// TwinCAT 3 PLC project Crane
// ProgramVersion: 3.1.4026.11
// libraries:
//   Tc2_Standard, * (Beckhoff Automation GmbH)
//   Tc2_System, * (Beckhoff Automation GmbH)
//   [Resi4MPM], * (Jan Wilch)
//   [xPPU], * (Jan Wilch)
// project tree:
//   / HardwareContainer.TcPOU, MAIN.TcPOU, PlcTask.TcTTO
// real-time tasks:
//   TASK PlcTask: cycle T#10ms, priority 20, ADS port 350
//   TASK PlcTask1: cycle T#10ms, priority 23, ADS port 351
//   TASK PlcTask2: cycle T#10ms, priority 22, ADS port 352
//   TASK PlcTask3: cycle T#10ms, priority 21, ADS port 353
// I/O:
//   DEVICE Device (EtherCAT), AmsNetId 192.168.82.13.3.1
//     Term 84 (EK1200) [EK1200-5000 EtherCAT Netzteil (2A E-Bus)]
//       Klemme 2 (EK1110) [EK1110 EtherCAT-Verlängerung]
//     BK1 (EK1100) [EK1100 EtherCAT-Koppler (2A E-Bus)]
//       1.2 (EL1004) [EL1004 4K. Dig. Eingang 24V, 3ms]
//       1.3 (EL1004) [EL1004 4K. Dig. Eingang 24V, 3ms]
//       1.4 (EL1004) [EL1004 4K. Dig. Eingang 24V, 3ms]
//       1.5 (EL1004) [EL1004 4K. Dig. Eingang 24V, 3ms]
//       1.6 (EL2004) [EL2004 4K. Dig. Ausgang 24V, 0.5A]
//       1.9 (EL2004) [EL2004 4K. Dig. Ausgang 24V, 0.5A]
//       1.10 (EL2004) [EL2004 4K. Dig. Ausgang 24V, 0.5A]
//       1.11 (EL2004) [EL2004 4K. Dig. Ausgang 24V, 0.5A]
//       1.12 (EL1004) [EL1004 4K. Dig. Eingang 24V, 3ms]
//       1.13 (EL3162) [EL3162 2K. Ana. Eingang 0-10V]
//       1.14 (EL9011) [EL9011 Endklemme]
//     BK2&3 (EK1100) [EK1100 EtherCAT-Koppler (2A E-Bus)]
//       2&3.2 (EL1004) [EL1004 4K. Dig. Eingang 24V, 3ms]
//       2&3.3 (EL1004) [EL1004 4K. Dig. Eingang 24V, 3ms]
//       2&3.4 (EL1004) [EL1004 4K. Dig. Eingang 24V, 3ms]
//       2&3.5 (EL1004) [EL1004 4K. Dig. Eingang 24V, 3ms]
//       2&3.6 (EL1004) [EL1004 4K. Dig. Eingang 24V, 3ms]
//       2&3.7 (EL1004) [EL1004 4K. Dig. Eingang 24V, 3ms]
//       2&3.10 (EL2004) [EL2004 4K. Dig. Ausgang 24V, 0.5A]
//       2&3.11 (EL2004) [EL2004 4K. Dig. Ausgang 24V, 0.5A]
//       2&3.12 (EL2004) [EL2004 4K. Dig. Ausgang 24V, 0.5A]
//       2&3.13 (EL2004) [EL2004 4K. Dig. Ausgang 24V, 0.5A]
//       2&3.14 (EL1004) [EL1004 4K. Dig. Eingang 24V, 3ms]
//       2&3.16 (EL4102) [EL4102 2K. Ana. Ausgang 0-10V]
//       2&3.17 (EL4102) [EL4102 2K. Ana. Ausgang 0-10V]
//       2&3.18 (EL9011) [EL9011 Endklemme]
//     BK4 (EK1100) [EK1100 EtherCAT-Koppler (2A E-Bus)]
//       4.2 (EL1808) [EL1808 8K. Dig. Eingang 24V, 3ms]
//       4.3 (EL1004) [EL1004 4K. Dig. Eingang 24V, 3ms]
//       4.4 (EL1004) [EL1004 4K. Dig. Eingang 24V, 3ms]
//       4.5 (EL1004) [EL1004 4K. Dig. Eingang 24V, 3ms]
//       4.6 (EL1004) [EL1004 4K. Dig. Eingang 24V, 3ms]
//       4.7 (EL1004) [EL1004 4K. Dig. Eingang 24V, 3ms]
//       4.8 (EL3064) [EL3064 4K.Ana. Eingang 0-10V]
//       4.9 (EL3064) [EL3064 4K.Ana. Eingang 0-10V]
//       4.10 (EL3164) [EL3164 4K. Ana. Eingang 0-10V]
//       4.11 (EL3054) [EL3054 4K.Ana. Eingang 4-20mA]
//       Klemme 90 (EL3058) [EL3058 8K. Ana. Eingang 4-20mA]
//       4.13 (EL2004) [EL2004 4K. Dig. Ausgang 24V, 0.5A]
//       4.14 (EL2004) [EL2004 4K. Dig. Ausgang 24V, 0.5A]
//       4.15 (EL9011) [EL9011 Endklemme]
//     BK5 (EK1100) [EK1100 EtherCAT Coupler (2A E-Bus)]
//       5.2 (EL1008) [EL1008 8Ch. Dig. Input 24V, 3ms]
//       5.3 (EL5152) [EL5152 2Ch. Inc. Encoder]
//       5.6 (EL2008) [EL2008 8Ch. Dig. Output 24V, 0.5A]
//       5.7 (EL4102) [EL4102 2Ch. Ana. Output 0-10V]
//       5.8 (EL9011) [EL9011 End Terminal]
//     BK6 (EK1100) [EK1100 EtherCAT Coupler (2A E-Bus)]
//       6.2 (EL3062) [EL3062 2Ch. Ana. Input 0-10V]
//       6.3 (EL6224) [EL6224 (IO Link Master)]
//       6.4 (EL9011) [EL9011 End Terminal]
//     BK7 (EK1100) [EK1100 EtherCAT Coupler (2A E-Bus)]
//       7.2 (EL1004) [EL1004 4Ch. Dig. Input 24V, 3ms]
//       7.5 (EL2004) [EL2004 4Ch. Dig. Output 24V, 0.5A]
//       7.8 (EL6224) [EL6224 (IO Link Master)]
//       7.9 (EL9011) [EL9011 End Terminal]
//     BK8 (EK1100) [EK1100 EtherCAT Coupler (2A E-Bus)]
//       8.2 (EL1008) [EL1008 8Ch. Dig. Input 24V, 3ms]
//       8.3 (EL1004) [EL1004 4Ch. Dig. Input 24V, 3ms]
//       8.4 (EL3062) [EL3062 2Ch. Ana. Input 0-10V]
//       8.5 (EL2004) [EL2004 4Ch. Dig. Output 24V, 0.5A]
//       8.8 (EL2008) [EL2008 8Ch. Dig. Output 24V, 0.5A]
//       8.9 (EL2004) [EL2004 4Ch. Dig. Output 24V, 0.5A]
//       Term 114 (EL1808) [EL1808 8Ch. Dig. Input 24V, 3ms]
//       8.10 (EL9011) [EL9011 End Terminal]
//     BK9 (EK1100) [EK1100 EtherCAT Coupler (2A E-Bus)]
//       9.2 (EL1004) [EL1004 4Ch. Dig. Input 24V, 3ms]
//       9.3 (EL5152) [EL5152 2Ch. Inc. Encoder]
//       9.6 (EL2004) [EL2004 4Ch. Dig. Output 24V, 0.5A]
//       9.7 (EL4102) [EL4102 2Ch. Ana. Output 0-10V]
//       9.8 (EL9011) [EL9011 End Terminal]
//     BK10 (EK1100) [EK1100 EtherCAT Coupler (2A E-Bus)]
//       10.2 (EL1004) [EL1004 4Ch. Dig. Input 24V, 3ms]
//       10.3 (EL5152) [EL5152 2Ch. Inc. Encoder]
//       10.6 (EL2004) [EL2004 4Ch. Dig. Output 24V, 0.5A]
//       10.7 (EL4102) [EL4102 2Ch. Ana. Output 0-10V]
//       10.8 (EL9011) [EL9011 End Terminal]
//     BK11 (EK1100) [EK1100 EtherCAT Coupler (2A E-Bus)]
//       11.2 (EL1004) [EL1004 4Ch. Dig. Input 24V, 3ms]
//       11.3 (EL3064) [EL3064 4Ch. Ana. Input 0-10V]
//       11.6 (EL2004) [EL2004 4Ch. Dig. Output 24V, 0.5A]
//       11.7 (EL9011) [EL9011 End Terminal]
// variable links:
//   Crane/Crane Instance <-> Device (EtherCAT)/BK1 (EK1100)/1.10 (EL2004)
//     PlcTask Outputs/MAIN.m_container.m_crane.Motor.DO_TurnClockwise <-> Channel 4/Output
//     PlcTask Outputs/MAIN.m_container.m_crane.Motor.DO_TurnCounterclockwise <-> Channel 3/Output
//   Crane/Crane Instance <-> Device (EtherCAT)/BK1 (EK1100)/1.13 (EL3162)
//     PlcTask Inputs/MAIN.m_container.m_crane.Motor.AI_Position <-> Channel 1/Value
//   Crane/Crane Instance <-> Device (EtherCAT)/BK1 (EK1100)/1.2 (EL1004)
//     PlcTask Inputs/MAIN.m_container.m_crane.o_VacuumGripper.DI_TakenIn <-> Channel 4/Input
//   Crane/Crane Instance <-> Device (EtherCAT)/BK1 (EK1100)/1.3 (EL1004)
//     PlcTask Inputs/MAIN.m_container.m_crane.o_MonostableCylinder.DI_Extended <-> Channel 1/Input
//     PlcTask Inputs/MAIN.m_container.m_crane.o_MonostableCylinder.DI_Retracted <-> Channel 2/Input
//   Crane/Crane Instance <-> Device (EtherCAT)/BK1 (EK1100)/1.4 (EL1004)
//     PlcTask Inputs/MAIN.m_container.m_crane.m_PresenceSensorAtConveyor.DI_WPDetected <-> Channel 4/Input
//     PlcTask Inputs/MAIN.m_container.m_crane.m_PresenceSensorAtStamp.DI_WPDetected <-> Channel 3/Input
//   Crane/Crane Instance <-> Device (EtherCAT)/BK1 (EK1100)/1.5 (EL1004)
//     PlcTask Inputs/MAIN.m_container.m_crane.m_PresenceSensorAtStack.DI_WPDetected <-> Channel 1/Input
//   Crane/Crane Instance <-> Device (EtherCAT)/BK1 (EK1100)/1.6 (EL2004)
//     PlcTask Outputs/MAIN.m_container.m_crane.o_VacuumGripper.DO_VacuumOn <-> Channel 1/Output
//   Crane/Crane Instance <-> Device (EtherCAT)/BK1 (EK1100)/1.9 (EL2004)
//     PlcTask Outputs/MAIN.m_container.m_crane.o_MonostableCylinder.DO_Extend <-> Channel 1/Output
//   Crane/Crane Instance <-> Device (EtherCAT)/BK4 (EK1100)/Term 90 (EL3058)
//     PlcTask Inputs/MAIN.m_container.m_crane.o_MonostableCylinder.AI_PositionTransmitter <-> AI Standard Channel 2/Value
//   Crane/Crane Instance <-> Device (EtherCAT)/BK5 (EK1100)/5.2 (EL1008)
//     PlcTask Inputs/MAIN.m_panelMgr.DI_ModeSwitch <-> Channel 3/Input
//     PlcTask Inputs/MAIN.m_panelMgr.DI_ResetBtn <-> Channel 4/Input
//     PlcTask Inputs/MAIN.m_panelMgr.DI_StartBtn <-> Channel 1/Input
//     PlcTask Inputs/MAIN.m_panelMgr.DI_StopBtn <-> Channel 2/Input
//   LargeSortingConveyor/LargeSortingConveyor Instance <-> Device (EtherCAT)/BK2&3 (EK1100)/2&3.11 (EL2004)
//     PlcTask Outputs/MAIN.m_container.m_LSC.Motor.DO_TurnClockwise <-> Channel 4/Output
//     PlcTask Outputs/MAIN.m_container.m_LSC.m_rampPusherMid.DO_Extend <-> Channel 3/Output
//     PlcTask Outputs/MAIN.m_container.m_LSC.m_rampPusherStart.DO_Extend <-> Channel 2/Output
//   LargeSortingConveyor/LargeSortingConveyor Instance <-> Device (EtherCAT)/BK2&3 (EK1100)/2&3.12 (EL2004)
//     PlcTask Outputs/MAIN.m_container.m_LSC.Motor.DO_TurnCounterclockwise <-> Channel 1/Output
//     PlcTask Outputs/MAIN.m_panelMgr.DO_GreenLight <-> Channel 2/Output
//     PlcTask Outputs/MAIN.m_panelMgr.DO_WhiteLight <-> Channel 3/Output
//   LargeSortingConveyor/LargeSortingConveyor Instance <-> Device (EtherCAT)/BK2&3 (EK1100)/2&3.3 (EL1004)
//     PlcTask Inputs/MAIN.m_panelMgr.DI_EStopBtn <-> Channel 3/Input
//     PlcTask Inputs/MAIN.m_panelMgr.DI_StartBtn <-> Channel 4/Input
//   LargeSortingConveyor/LargeSortingConveyor Instance <-> Device (EtherCAT)/BK2&3 (EK1100)/2&3.4 (EL1004)
//     PlcTask Inputs/MAIN.m_container.m_LSC.m_inductiveSensorStart.DI_WPMetallic <-> Channel 4/Input
//     PlcTask Inputs/MAIN.m_container.m_LSC.m_opticalSensorStart.DI_WPLight <-> Channel 2/Input
//     PlcTask Inputs/MAIN.m_container.m_LSC.m_presenceSensorStart.DI_WPDetected <-> Channel 3/Input
//     PlcTask Inputs/MAIN.m_panelMgr.DI_ModeSwitch <-> Channel 1/Input
//   LargeSortingConveyor/LargeSortingConveyor Instance <-> Device (EtherCAT)/BK2&3 (EK1100)/2&3.5 (EL1004)
//     PlcTask Inputs/MAIN.m_container.m_LSC.m_inductiveSensorMid.DI_WPMetallic <-> Channel 2/Input
//     PlcTask Inputs/MAIN.m_container.m_LSC.m_opticalSensorEnd.DI_WPLight <-> Channel 3/Input
//     PlcTask Inputs/MAIN.m_container.m_LSC.m_opticalSensorMid.DI_WPLight <-> Channel 1/Input
//   LargeSortingConveyor/LargeSortingConveyor Instance <-> Device (EtherCAT)/BK2&3 (EK1100)/2&3.6 (EL1004)
//     PlcTask Inputs/MAIN.m_container.m_LSC.m_rampPusherMid.DI_Extended <-> Channel 3/Input
//     PlcTask Inputs/MAIN.m_container.m_LSC.m_rampPusherMid.DI_Retracted <-> Channel 4/Input
//     PlcTask Inputs/MAIN.m_container.m_LSC.m_rampPusherStart.DI_Extended <-> Channel 1/Input
//     PlcTask Inputs/MAIN.m_container.m_LSC.m_rampPusherStart.DI_Retracted <-> Channel 2/Input
//   LargeSortingConveyor/LargeSortingConveyor Instance <-> Device (EtherCAT)/BK4 (EK1100)/4.2 (EL1808)
//     PlcTask Inputs/MAIN.m_container.m_LSC.m_rampEnd.m_presenceSensorRampFull.DI_WPDetected <-> Channel 8/Input
//     PlcTask Inputs/MAIN.m_container.m_LSC.m_rampMiddle.m_presenceSensorRampFull.DI_WPDetected <-> Channel 7/Input
//     PlcTask Inputs/MAIN.m_container.m_LSC.m_rampStart.m_presenceSensorRampFull.DI_WPDetected <-> Channel 6/Input
//   LargeSortingConveyor/LargeSortingConveyor Instance <-> Device (EtherCAT)/BK4 (EK1100)/Term 90 (EL3058)
//     PlcTask Inputs/MAIN.m_container.m_LSC.m_rampPusherMid.AI_PositionTransmitter <-> AI Standard Channel 5/Value
//     PlcTask Inputs/MAIN.m_container.m_LSC.m_rampPusherStart.AI_PositionTransmitter <-> AI Standard Channel 6/Value
//   LargeSortingConveyor/LargeSortingConveyor Instance <-> Device (EtherCAT)/BK7 (EK1100)/7.2 (EL1004)
//     PlcTask Inputs/MAIN.m_container.m_LSC.m_Switch.DI_Extended <-> Channel 4/Input
//     PlcTask Inputs/MAIN.m_container.m_LSC.m_Switch.DI_Retracted <-> Channel 3/Input
//   LargeSortingConveyor/LargeSortingConveyor Instance <-> Device (EtherCAT)/BK7 (EK1100)/7.5 (EL2004)
//     PlcTask Outputs/MAIN.m_container.m_LSC.m_Switch.DO_Extend <-> Channel 3/Output
//   Stack/Stack Instance <-> Device (EtherCAT)/BK1 (EK1100)/1.10 (EL2004)
//     PlcTask Outputs/MAIN.m_panelMgr.DO_GreenLight <-> Channel 1/Output
//     PlcTask Outputs/MAIN.m_panelMgr.DO_WhiteLight <-> Channel 2/Output
//   Stack/Stack Instance <-> Device (EtherCAT)/BK1 (EK1100)/1.2 (EL1004)
//     PlcTask Inputs/MAIN.m_panelMgr.DI_EStopBtn <-> Channel 1/Input
//     PlcTask Inputs/MAIN.m_panelMgr.DI_ModeSwitch <-> Channel 3/Input
//     PlcTask Inputs/MAIN.m_panelMgr.DI_StartBtn <-> Channel 2/Input
//   Stack/Stack Instance <-> Device (EtherCAT)/BK1 (EK1100)/1.3 (EL1004)
//     PlcTask Inputs/MAIN.m_container.m_stack.o_slidingCylinder.DI_Extended <-> Channel 4/Input
//     PlcTask Inputs/MAIN.m_container.m_stack.o_slidingCylinder.DI_Retracted <-> Channel 3/Input
//   Stack/Stack Instance <-> Device (EtherCAT)/BK1 (EK1100)/1.4 (EL1004)
//     PlcTask Inputs/MAIN.m_container.m_stack.m_Inductivesensor.DI_WPMetallic <-> Channel 1/Input
//     PlcTask Inputs/MAIN.m_container.m_stack.m_Opticalsensor.DI_WPLight <-> Channel 2/Input
//   Stack/Stack Instance <-> Device (EtherCAT)/BK1 (EK1100)/1.5 (EL1004)
//     PlcTask Inputs/MAIN.m_container.m_stack.m_Presencesensor.DI_WPDetected <-> Channel 2/Input
//   Stack/Stack Instance <-> Device (EtherCAT)/BK1 (EK1100)/1.9 (EL2004)
//     PlcTask Outputs/MAIN.m_container.m_stack.o_slidingCylinder.DO_Extend <-> Channel 2/Output
//   Stack/Stack Instance <-> Device (EtherCAT)/BK4 (EK1100)/4.3 (EL1004)
//     PlcTask Inputs/MAIN.m_container.m_stack.o_slidingCylinder.DI_BoundaryPressure <-> Channel 1/Input
//   Stack/Stack Instance <-> Device (EtherCAT)/BK6 (EK1100)/6.2 (EL3062)
//     PlcTask Inputs/MAIN.m_container.m_stack.m_Weightsensor.AI_WPWeight <-> AI Standard Channel 1/Value
//   Stamp/Stamp Instance <-> Device (EtherCAT)/BK2&3 (EK1100)/2&3.10 (EL2004)
//     PlcTask Outputs/MAIN.m_container.m_stamp.m_slidingCylinder.DO_Extend <-> Channel 1/Output
//     PlcTask Outputs/MAIN.m_container.m_stamp.m_slidingCylinder.DO_Retract <-> Channel 2/Output
//     PlcTask Outputs/MAIN.m_container.m_stamp.m_stampingCylinder.DO_Extend <-> Channel 3/Output
//     PlcTask Outputs/MAIN.m_panelMgr.DO_GreenLight <-> Channel 4/Output
//   Stamp/Stamp Instance <-> Device (EtherCAT)/BK2&3 (EK1100)/2&3.11 (EL2004)
//     PlcTask Outputs/MAIN.m_panelMgr.DO_WhiteLight <-> Channel 1/Output
//   Stamp/Stamp Instance <-> Device (EtherCAT)/BK2&3 (EK1100)/2&3.16 (EL4102)
//     PlcTask Outputs/MAIN.m_container.m_stamp.m_pressureValve.AO_SetPressure <-> Channel 2/Output
//   Stamp/Stamp Instance <-> Device (EtherCAT)/BK2&3 (EK1100)/2&3.2 (EL1004)
//     PlcTask Inputs/MAIN.m_container.m_stamp.m_slidingCylinder.DI_Extended <-> Channel 2/Input
//     PlcTask Inputs/MAIN.m_container.m_stamp.m_slidingCylinder.DI_Retracted <-> Channel 3/Input
//     PlcTask Inputs/MAIN.m_container.m_stamp.m_stampingCylinder.DI_Retracted <-> Channel 4/Input
//     PlcTask Inputs/MAIN.m_panelMgr.DI_ModeSwitch <-> Channel 1/Input
//   Stamp/Stamp Instance <-> Device (EtherCAT)/BK2&3 (EK1100)/2&3.3 (EL1004)
//     PlcTask Inputs/MAIN.m_container.m_stamp.m_presenceSensor.DI_WPDetected <-> Channel 2/Input
//     PlcTask Inputs/MAIN.m_container.m_stamp.m_stampingCylinder.DI_Extended <-> Channel 1/Input
//   Stamp/Stamp Instance <-> Device (EtherCAT)/BK2&3 (EK1100)/2&3.7 (EL1004)
//     PlcTask Inputs/MAIN.m_panelMgr.DI_EStopBtn <-> Channel 3/Input
//     PlcTask Inputs/MAIN.m_panelMgr.DI_StartBtn <-> Channel 4/Input
//   Stamp/Stamp Instance <-> Device (EtherCAT)/BK4 (EK1100)/4.3 (EL1004)
//     PlcTask Inputs/MAIN.m_container.m_stamp.m_slidingCylinder.DI_BoundaryPressure <-> Channel 2/Input
//   Stamp/Stamp Instance <-> Device (EtherCAT)/BK4 (EK1100)/4.4 (EL1004)
//     PlcTask Inputs/MAIN.m_container.m_stamp.m_stampingCylinder.DI_BoundaryPressure <-> Channel 4/Input
//   Stamp/Stamp Instance <-> Device (EtherCAT)/BK4 (EK1100)/4.6 (EL1004)
//     PlcTask Inputs/MAIN.m_container.m_stamp.m_stampingCylinder.DI_BoundaryFlowPressure <-> Channel 1/Input
//   Stamp/Stamp Instance <-> Device (EtherCAT)/BK4 (EK1100)/4.9 (EL3064)
//     PlcTask Inputs/MAIN.m_container.m_stamp.m_stampingCylinder.AI_PressureSensor <-> AI Standard Channel 2/Value
//   Stamp/Stamp Instance <-> Device (EtherCAT)/BK4 (EK1100)/Term 90 (EL3058)
//     PlcTask Inputs/MAIN.m_container.m_stamp.m_slidingCylinder.AI_PositionTransmitter <-> AI Standard Channel 3/Value
//     PlcTask Inputs/MAIN.m_container.m_stamp.m_stampingCylinder.AI_PositionTransmitter <-> AI Standard Channel 4/Value

CONFIGURATION Crane
    RESOURCE PLC ON TwinCAT3
        TASK PlcTask(INTERVAL := T#10ms, PRIORITY := 21);
        PROGRAM MAIN WITH PlcTask : MAIN;
    END_RESOURCE
END_CONFIGURATION

// ---- MAIN.TcPOU
PROGRAM MAIN
VAR CONSTANT
	IGNORE_DEFINITION: BOOL := TRUE;
END_VAR
VAR
	m_errorManager: ErrorManager;
	m_services: ServiceContainer(ADR(m_errorManager));
	
	// the Safety Door is assigned to the Crane
	m_panelMgr: PanelManager(
		m_services.PtrStateTracker,
		EProcessVariables.Pnl_Door_Start, 
		EProcessVariables.Pnl_Door_Stop, 
		EProcessVariables.Pnl_Door_Mode, 
		0, 
		EProcessVariables.Pnl_Door_Reset);
	
	// instantiate machine behavior model
	m_container: HardwareContainer(
		m_services.PtrStateTracker, 
		m_services.PtrProcessManager, 
		ADR(m_errorManager));
	
	m_modes: MachineModes(ADR(m_services), ADR(m_panelMgr));
	
	m_appObservation: ARRAY[EProcessVariables.OpMode_Crane..EProcessVariables.OpMode_Crane] OF SValue;

	// TESTING
// 	m_testCopyFromStack: BOOL;
// 	m_testCopyToStamp: BOOL;
// 	m_testCopyFromStamp: BOOL;
// 	m_rtFromStack: R_TRIG;
// 	m_rtToStamp: R_TRIG;
// 	m_rtFromStamp: R_TRIG;
// 	m_fromStackBusy: BOOL;
// 	m_toStampBusy: BOOL;
// 	m_fromStampBusy: BOOL;
// 	m_cycCount: UINT;
// 	
// 	m_lscConnected: BOOL;
// 	m_craneConnected: BOOL;
// 	m_stackConnected: BOOL;
// 	m_stampConnected: BOOL;
END_VAR

// process state observation
m_appObservation[EProcessVariables.OpMode_Crane].DataType := EDataType.string_t;
m_appObservation[EProcessVariables.OpMode_Crane].Value.String_t := m_modes.SFCCurrentStep;
m_appObservation[EProcessVariables.OpMode_Crane].Defined := TRUE;

// cylic service updates
m_services.PtrStateTracker^.CyclicUpdateStatus(IGNORE_DEFINITION, m_appObservation);
m_services.PtrProcessManager^.CyclicManageBehavior();

// main state machine
m_modes();

// TESTING (shift register)
// m_rtFromStack(CLK := m_testCopyFromStack);
// m_rtToStamp(CLK := m_testCopyToStamp);
// m_rtFromStamp(CLK := m_testCopyFromStamp);
// IF m_rtFromStack.Q OR m_fromStackBusy THEN	
// 	m_fromStackBusy := NOT m_services.PtrStateTracker^.ShiftProduct(EProducts.stack_product, EProducts.crane_product);
// 	m_cycCount := m_cycCount + 1;
// END_IF
// IF m_rtToStamp.Q OR m_toStampBusy THEN
// 	m_toStampBusy := NOT m_services.PtrStateTracker^.ShiftProduct(EProducts.crane_product, EProducts.stamp_product);
// 	m_cycCount := m_cycCount + 1;
// END_IF
// IF m_rtFromStamp.Q OR m_fromStampBusy THEN
// 	m_fromStampBusy := NOT m_services.PtrStateTracker^.ShiftProduct(EProducts.stamp_product, EProducts.crane_product);
// 	m_cycCount := m_cycCount + 1;
// END_IF
// IF NOT m_testCopyFromStack AND NOT m_testCopyFromStamp AND NOT m_testCopyToStamp THEN
// 	m_cycCount := 0;
// END_IF

// TESTING
// IF m_services.PtrStateTracker^.GetString(EProcessVariables.OpMode_LSC) <> '' THEN
// 	m_lscConnected := TRUE;
// END_IF
// IF m_services.PtrStateTracker^.GetString(EProcessVariables.OpMode_Stack) <> '' THEN
// 	m_stackConnected := TRUE;
// END_IF
// IF m_services.PtrStateTracker^.GetString(EProcessVariables.OpMode_Stamp) <> '' THEN
// 	m_stampConnected := TRUE;
// END_IF
// IF m_services.PtrStateTracker^.GetString(EProcessVariables.OpMode_Crane) <> '' THEN
// 	m_craneConnected := TRUE;
// END_IF

END_PROGRAM

// ---- HardwareContainer.TcPOU
FUNCTION_BLOCK HardwareContainer
VAR
	// hardware control POUs
	m_crane: Crane;
	m_indic: ActivityIndicator(i_signalProcVar := EProcessVariables.Test_CraneFree);
	
	// products
	{attribute 'OPC.UA.DA' := '1'}
	{attribute 'OPC.UA.DA.Access' := '1'}
	m_craneWP: xPPUProduct(EProcessVariables.Crane_ProductType, EProcessVariables.Crane_ProductStamped);
	
	// hardware observation (if not included in hardware control)
	m_observeCrane: ObserveCrane(ADR(m_crane), ADR(m_craneWP));
	
	// control primitives
	m_craneMoveToStack: Crane_MoveToStack(ADR(m_crane));
	m_craneMoveToStamp: Crane_MoveToStamp(ADR(m_crane));
	m_craneMoveToLSC: Crane_MoveToLSC(ADR(m_crane));
	m_cranePickUpWP: Crane_PickUpWP(ADR(m_crane));
	m_cranePutDownWP: Crane_PutDownWP(ADR(m_crane));
	
	m_delay: Delay;
	m_indicCP_Crane: IndicateActivity(i_id := EPrimitives.Gen_IndicateActive_Crane, i_ptrIndicator := ADR(m_indic));
	m_forceVal_Crane: ForceProcessVariable(i_id := EPrimitives.Gen_ForceVariable_Crane);
	
	// module sequences
END_VAR

METHOD FB_init : BOOL
VAR_INPUT
	bInitRetains : BOOL; // if TRUE, the retain variables are initialized (warm start / cold start)
	bInCopyCode : BOOL;  // if TRUE, the instance afterwards gets moved into the copy code (online change)

	i_ptrStateTracker: POINTER TO StateTracker;
	i_ptrProcessManager: POINTER TO ProcessManager;
	
	i_ptrErrorManager: POINTER TO ErrorManagerBase;
END_VAR
m_craneMoveToStack.ProvideServices(i_ptrProcessManager, i_ptrStateTracker);
m_craneMoveToStamp.ProvideServices(i_ptrProcessManager, i_ptrStateTracker);
m_craneMoveToLSC.ProvideServices(i_ptrProcessManager, i_ptrStateTracker);
m_cranePickUpWP.ProvideServices(i_ptrProcessManager, i_ptrStateTracker);
m_cranePutDownWP.ProvideServices(i_ptrProcessManager, i_ptrStateTracker);

m_delay.ProvideServices(i_ptrProcessManager, i_ptrStateTracker);
m_indicCP_Crane.ProvideServices(i_ptrProcessManager, i_ptrStateTracker);
m_forceVal_Crane.ProvideServices(i_ptrProcessManager, i_ptrStateTracker);

// provide Behaviors to the Process Manager
i_ptrProcessManager^.AddPrimitive(ADR(m_craneMoveToStack));
i_ptrProcessManager^.AddPrimitive(ADR(m_craneMoveToStamp));
i_ptrProcessManager^.AddPrimitive(ADR(m_craneMoveToLSC));
i_ptrProcessManager^.AddPrimitive(ADR(m_cranePickUpWP));
i_ptrProcessManager^.AddPrimitive(ADR(m_cranePutDownWP));

i_ptrProcessManager^.AddPrimitive(ADR(m_delay));
i_ptrProcessManager^.AddPrimitive(ADR(m_indicCP_Crane));
i_ptrProcessManager^.AddPrimitive(ADR(m_forceVal_Crane));

// provide observations to the Process Manager
i_ptrStateTracker^.AddObservation(ADR(m_observeCrane));
i_ptrStateTracker^.AddObservation(ADR(m_indic));

// provide workpieces to the Process Manager
i_ptrStateTracker^.RegisterLocalProduct(EProducts.crane_product, ADR(m_craneWP));
END_METHOD

END_FUNCTION_BLOCK
